ABB RobotStudio station: DigitalTwin.rsstnx

Station DigitalTwin (saved by RobotStudio 22.2.10013.1)
Controller CRB15000_5_95
  mechanical unit ROB_1: CRB15000_5_95__02, 6 joints, base frame (0, 0, 0) mm
Layout (positions relative to the parent item):
  - CRB15000_5_95__02 [mechanism, from Robots\CRB15000_5_95__02.rslib] at (0, 0, 0) mm; joint values [0.1831, -0.1768, 0.4028, -0.1676, 0.7382, 1.3507] (rad or m)
  - gripper_rg6 [part] at (519.39, 94.7, 666.71) mm, rotated rx 147.83 ry 16.31 rz 113.46 deg, size 75.5 x 155 x 263.6 mm
Attachment: gripper_rg6 is attached to CRB15000_5_95__02 / Link6
